// TIA Portal V16 export
// export: Created 2021-03-05T14:22:10.5832866Z, ExportSetting WithDefaults, DisplayName Totally Integrated Automation Portal, DisplayVersion V16, DisplayName TIA Portal Version Control Interface, DisplayVersion V16, DisplayName TIA Portal Openness, DisplayVersion V16, DisplayName SINAMICS Startdrive Advanced, DisplayVersion V16, DisplayName SINAMICS Startdrive G130, G150, S120, S150, SINAMICS MV, S210, DisplayVersion V16, DisplayName SINAMICS Startdrive G110M, G120, G120C, G120D, G120P, DisplayVersion V16, DisplayName STEP 7 Professional, DisplayVersion V16, DisplayName STEP 7 Safety, DisplayVersion V16, DisplayName WinCC Professional, DisplayVersion V16
FUNCTION_BLOCK "fbMain"   // FB2, LAD
{ S7_Optimized_Access := 'TRUE' }
VERSION : 0.1
// stored: AutoNumber true, IsIECCheckEnabled false, IsRetainMemResEnabled false, MemoryReserve 100, SetENOAutomatically false, UDAEnableTagReadback false
   VAR
      Room { ExternalVisible := 'False'} : Array[1.."MAX_ROOMS"] of "fbRoom";
      Config { S7_SetPoint := 'True'} : "fbConfig";
   END_VAR
   VAR_TEMP
      iRoomCount : Int;
      iRackCount : Int;
      iPos : DInt;
   END_VAR
   // Config.iNumRooms := 0;
BEGIN

REGION Network 1 (SCL)
   // bInSimulation := TRUE skips IO device configuration steps
   #Config(bInSimulation := #Config.bInSimulation);
END_REGION

REGION Network 2 (SCL)
   #Room[1].Rack[1].Fertigation.ShelvesFertigation[1].DI_Level_Switch.bStatus := "DI_Level_SW_R1S1";
   #Room[1].Rack[1].Fertigation.ShelvesFertigation[2].DI_Level_Switch.bStatus := "DI_Level_SW_R1S2";
   #Room[1].Rack[1].Fertigation.ShelvesFertigation[3].DI_Level_Switch.bStatus := "DI_Level_SW_R1S3";
   #Room[1].Rack[1].Fertigation.ShelvesFertigation[4].DI_Level_Switch.bStatus := "DI_Level_SW_R1S4";
   #Room[1].Rack[1].Fertigation.ShelvesFertigation[5].DI_Level_Switch.bStatus := "DI_Level_SW_R1S5";
   #Room[1].Rack[1].Fertigation.ShelvesFertigation[6].DI_Level_Switch.bStatus := "DI_Level_SW_R1S6";

   #Room[1].Rack[2].Fertigation.ShelvesFertigation[1].DI_Level_Switch.bStatus := "DI_Level_SW_R2S1";
   #Room[1].Rack[2].Fertigation.ShelvesFertigation[2].DI_Level_Switch.bStatus := "DI_Level_SW_R2S2";
   #Room[1].Rack[2].Fertigation.ShelvesFertigation[3].DI_Level_Switch.bStatus := "DI_Level_SW_R2S3";
   #Room[1].Rack[2].Fertigation.ShelvesFertigation[4].DI_Level_Switch.bStatus := "DI_Level_SW_R2S4";
   #Room[1].Rack[2].Fertigation.ShelvesFertigation[5].DI_Level_Switch.bStatus := "DI_Level_SW_R2S5";
   #Room[1].Rack[2].Fertigation.ShelvesFertigation[6].DI_Level_Switch.bStatus := "DI_Level_SW_R2S6";

   #Room[1].Rack[3].Fertigation.ShelvesFertigation[1].DI_Level_Switch.bStatus := "DI_Level_SW_R3S1";
   #Room[1].Rack[3].Fertigation.ShelvesFertigation[2].DI_Level_Switch.bStatus := "DI_Level_SW_R3S2";
   #Room[1].Rack[3].Fertigation.ShelvesFertigation[3].DI_Level_Switch.bStatus := "DI_Level_SW_R3S3";
   #Room[1].Rack[3].Fertigation.ShelvesFertigation[4].DI_Level_Switch.bStatus := "DI_Level_SW_R3S4";
   #Room[1].Rack[3].Fertigation.ShelvesFertigation[5].DI_Level_Switch.bStatus := "DI_Level_SW_R3S5";
   #Room[1].Rack[3].Fertigation.ShelvesFertigation[6].DI_Level_Switch.bStatus := "DI_Level_SW_R3S6";

   #Room[1].Rack[4].Fertigation.ShelvesFertigation[1].DI_Level_Switch.bStatus := "DI_Level_SW_R4S1";
   #Room[1].Rack[4].Fertigation.ShelvesFertigation[2].DI_Level_Switch.bStatus := "DI_Level_SW_R4S2";
   #Room[1].Rack[4].Fertigation.ShelvesFertigation[3].DI_Level_Switch.bStatus := "DI_Level_SW_R4S3";
   #Room[1].Rack[4].Fertigation.ShelvesFertigation[4].DI_Level_Switch.bStatus := "DI_Level_SW_R4S4";
   #Room[1].Rack[4].Fertigation.ShelvesFertigation[5].DI_Level_Switch.bStatus := "DI_Level_SW_R4S5";
   #Room[1].Rack[4].Fertigation.ShelvesFertigation[6].DI_Level_Switch.bStatus := "DI_Level_SW_R4S6";
END_REGION

REGION Network 3 (SCL)
   #Room[1].Rack[1].Fertigation.arrAI[1] := "Rack_1_Reservoir_Level";
   #Room[1].Rack[2].Fertigation.arrAI[1] := "Rack_2_Reservoir_Level";
   #Room[1].Rack[3].Fertigation.arrAI[1] := "Rack_3_Reservoir_Level";
   #Room[1].Rack[4].Fertigation.arrAI[1] := "Rack_4_Reservoir_Level";
END_REGION

REGION Network 4 (SCL): Map AI input array to all room and rack inputs
   (*
   IF #Config.Status.bDone THEN

       FOR #iRoomCount := 1 TO UINT_TO_INT("MAX_ROOMS") DO

           #iPos := 1; // input array is 1 indexed

           MOVE_BLK(IN := "GlobalAI".Room[#iRoomCount].AI[#iPos],
                    COUNT := "NUM_AI_ROOM",
                    OUT => #Room[#iRoomCount].arrAI[1]);

           #iPos += "NUM_AI_ROOM";


           FOR #iRackCount := 1 TO UINT_TO_INT("MAX_RACKS_PER_ROOM") DO

               MOVE_BLK(IN := "GlobalAI".Room[#iRoomCount].AI[#iPos],
                        COUNT := "NUM_AI_RACK",
                        OUT => #Room[#iRoomCount].Rack[#iRackCount].arrAI[1]);

               #iPos += "NUM_AI_RACK";

           END_FOR;

           #iPos += "EXTRA_AI_PER_ROOM"; // skip over unused points

       END_FOR;

   END_IF;
   *)
END_REGION

REGION Network 5 (SCL): Map DI input array to all room and rack inputs
   (*
   IF #Config.Status.bDone THEN

       FOR #iRoomCount := 1 TO UINT_TO_INT("MAX_ROOMS") DO

           #iPos := 1; // input array is 1 indexed

           (*
           MOVE_BLK(IN := "GlobalDI".Room[#iRoomCount].DI[#iPos],
                    COUNT := "MAX_DI_ROOM",
                    OUT => #Room[#iRoomCount].DI_Level_Switch.bStatus);
           *) 

           #iPos += "NUM_AI_ROOM";

           (*
           FOR #iRackCount := 1 TO UINT_TO_INT("MAX_RACKS_PER_ROOM") DO

               MOVE_BLK(IN := "GlobalDI".Room[#iRoomCount].DI[#iPos],
                        COUNT := "NUM_DI_RACK",
                        OUT => #Room[#iRoomCount].Rack[#iRackCount].arrDI[1]);

               #iPos += "NUM_AI_RACK";

           END_FOR;
           *)

           #iPos += "EXTRA_AI_PER_ROOM"; // skip over unused points

       END_FOR;

   END_IF;*)
END_REGION

REGION Network 6 (SCL): Call FBs for all configured rooms
   IF #Config.Status.bDone THEN

       FOR #iRoomCount := 1 TO #Config.iNumRooms DO

           #Room[#iRoomCount](arrAI := #Room[#iRoomCount].arrAI);

       END_FOR;

   END_IF;
END_REGION

REGION Network 7 (SCL): Combine all room and rack outputs into a single output array
   (*
   IF #Config.Status.bDone THEN

       FOR #iRoomCount := 1 TO UINT_TO_INT("MAX_ROOMS") DO

           #iPos := 1; // output array is 1 indexed

           MOVE_BLK(IN := #Room[#iRoomCount].arrDQ[1],
                    COUNT := "NUM_DQ_ROOM",
                    OUT => "GlobalDQ".Room[#iRoomCount].DQ[#iPos]);

           #iPos += "NUM_DQ_ROOM";


           FOR #iRackCount := 1 TO UINT_TO_INT("MAX_RACKS_PER_ROOM") DO

               MOVE_BLK(IN := #Room[#iRoomCount].Rack[#iRackCount].arrDQ[1],
                        COUNT := "NUM_DQ_RACK",
                        OUT => "GlobalDQ".Room[#iRoomCount].DQ[#iPos]);

               #iPos += "NUM_DQ_RACK";

           END_FOR;

           #iPos += "EXTRA_DQ_PER_ROOM"; // skip over unused points

       END_FOR;

   END_IF;
   *)
END_REGION

REGION Network 8 (SCL)
   "Rack_1_RO" := #Room[1].Rack[1].Fertigation.arrDQ[1];
   "Rack_1_Discharge" := #Room[1].Rack[1].Fertigation.arrDQ[2];

   "Rack_1_Shelf_1_Fill" := #Room[1].Rack[1].Fertigation.ShelvesFertigation[1].arrDQ[1];
   "Rack_1_Shelf_1_Drain" := #Room[1].Rack[1].Fertigation.ShelvesFertigation[1].arrDQ[2];
   "Rack_1_Shelf_2_Fill" := #Room[1].Rack[1].Fertigation.ShelvesFertigation[2].arrDQ[1];
   "Rack_1_Shelf_2_Drain" := #Room[1].Rack[1].Fertigation.ShelvesFertigation[2].arrDQ[2];
   "Rack_1_Shelf_3_Fill" := #Room[1].Rack[1].Fertigation.ShelvesFertigation[3].arrDQ[1];
   "Rack_1_Shelf_3_Drain" := #Room[1].Rack[1].Fertigation.ShelvesFertigation[3].arrDQ[2];
   "Rack_1_Shelf_4_Fill" := #Room[1].Rack[1].Fertigation.ShelvesFertigation[4].arrDQ[1];
   "Rack_1_Shelf_4_Drain" := #Room[1].Rack[1].Fertigation.ShelvesFertigation[4].arrDQ[2];
   "Rack_1_Shelf_5_Fill" := #Room[1].Rack[1].Fertigation.ShelvesFertigation[5].arrDQ[1];
   "Rack_1_Shelf_5_Drain" := #Room[1].Rack[1].Fertigation.ShelvesFertigation[5].arrDQ[2];
   "Rack_1_Shelf_6_Fill" := #Room[1].Rack[1].Fertigation.ShelvesFertigation[6].arrDQ[1];
   "Rack_1_Shelf_6_Drain" := #Room[1].Rack[1].Fertigation.ShelvesFertigation[6].arrDQ[2];

   "Rack_2_RO" := #Room[1].Rack[2].Fertigation.arrDQ[1];
   "Rack_2_Discharge" := #Room[1].Rack[2].Fertigation.arrDQ[2];

   "Rack_2_Shelf_1_Fill" := #Room[1].Rack[2].Fertigation.ShelvesFertigation[1].arrDQ[1];
   "Rack_2_Shelf_1_Drain" := #Room[1].Rack[2].Fertigation.ShelvesFertigation[1].arrDQ[2];
   "Rack_2_Shelf_2_Fill" := #Room[1].Rack[2].Fertigation.ShelvesFertigation[2].arrDQ[1];
   "Rack_2_Shelf_2_Drain" := #Room[1].Rack[2].Fertigation.ShelvesFertigation[2].arrDQ[2];
   "Rack_2_Shelf_3_Fill" := #Room[1].Rack[2].Fertigation.ShelvesFertigation[3].arrDQ[1];
   "Rack_2_Shelf_3_Drain" := #Room[1].Rack[2].Fertigation.ShelvesFertigation[3].arrDQ[2];
   "Rack_2_Shelf_4_Fill" := #Room[1].Rack[2].Fertigation.ShelvesFertigation[4].arrDQ[1];
   "Rack_2_Shelf_4_Drain" := #Room[1].Rack[2].Fertigation.ShelvesFertigation[4].arrDQ[2];
   "Rack_2_Shelf_5_Fill" := #Room[1].Rack[2].Fertigation.ShelvesFertigation[5].arrDQ[1];
   "Rack_2_Shelf_5_Drain" := #Room[1].Rack[2].Fertigation.ShelvesFertigation[5].arrDQ[2];
   "Rack_2_Shelf_6_Fill" := #Room[1].Rack[2].Fertigation.ShelvesFertigation[6].arrDQ[1];
   "Rack_2_Shelf_6_Drain" := #Room[1].Rack[2].Fertigation.ShelvesFertigation[6].arrDQ[2];


   "Rack_3_RO" := #Room[1].Rack[3].Fertigation.arrDQ[1];
   "Rack_3_Discharge" := #Room[1].Rack[3].Fertigation.arrDQ[2];

   "Rack_3_Shelf_1_Fill" := #Room[1].Rack[3].Fertigation.ShelvesFertigation[1].arrDQ[1];
   "Rack_3_Shelf_1_Drain" := #Room[1].Rack[3].Fertigation.ShelvesFertigation[1].arrDQ[2];
   "Rack_3_Shelf_2_Fill" := #Room[1].Rack[3].Fertigation.ShelvesFertigation[2].arrDQ[1];
   "Rack_3_Shelf_2_Drain" := #Room[1].Rack[3].Fertigation.ShelvesFertigation[2].arrDQ[2];
   "Rack_3_Shelf_3_Fill" := #Room[1].Rack[3].Fertigation.ShelvesFertigation[3].arrDQ[1];
   "Rack_3_Shelf_3_Drain" := #Room[1].Rack[3].Fertigation.ShelvesFertigation[3].arrDQ[2];
   "Rack_3_Shelf_4_Fill" := #Room[1].Rack[3].Fertigation.ShelvesFertigation[4].arrDQ[1];
   "Rack_3_Shelf_4_Drain" := #Room[1].Rack[3].Fertigation.ShelvesFertigation[4].arrDQ[2];
   "Rack_3_Shelf_5_Fill" := #Room[1].Rack[3].Fertigation.ShelvesFertigation[5].arrDQ[1];
   "Rack_3_Shelf_5_Drain" := #Room[1].Rack[3].Fertigation.ShelvesFertigation[5].arrDQ[2];
   "Rack_3_Shelf_6_Fill" := #Room[1].Rack[3].Fertigation.ShelvesFertigation[6].arrDQ[1];
   "Rack_3_Shelf_6_Drain" := #Room[1].Rack[3].Fertigation.ShelvesFertigation[6].arrDQ[2];

   "Rack_4_RO" := #Room[1].Rack[4].Fertigation.arrDQ[1];
   "Rack_4_Discharge" := #Room[1].Rack[4].Fertigation.arrDQ[2];

   "Rack_4_Shelf_1_Fill" := #Room[1].Rack[4].Fertigation.ShelvesFertigation[1].arrDQ[1];
   "Rack_4_Shelf_1_Drain" := #Room[1].Rack[4].Fertigation.ShelvesFertigation[1].arrDQ[2];
   "Rack_4_Shelf_2_Fill" := #Room[1].Rack[4].Fertigation.ShelvesFertigation[2].arrDQ[1];
   "Rack_4_Shelf_2_Drain" := #Room[1].Rack[4].Fertigation.ShelvesFertigation[2].arrDQ[2];
   "Rack_4_Shelf_3_Fill" := #Room[1].Rack[4].Fertigation.ShelvesFertigation[3].arrDQ[1];
   "Rack_4_Shelf_3_Drain" := #Room[1].Rack[4].Fertigation.ShelvesFertigation[3].arrDQ[2];
   "Rack_4_Shelf_4_Fill" := #Room[1].Rack[4].Fertigation.ShelvesFertigation[4].arrDQ[1];
   "Rack_4_Shelf_4_Drain" := #Room[1].Rack[4].Fertigation.ShelvesFertigation[4].arrDQ[2];
   "Rack_4_Shelf_5_Fill" := #Room[1].Rack[4].Fertigation.ShelvesFertigation[5].arrDQ[1];
   "Rack_4_Shelf_5_Drain" := #Room[1].Rack[4].Fertigation.ShelvesFertigation[5].arrDQ[2];
   "Rack_4_Shelf_6_Fill" := #Room[1].Rack[4].Fertigation.ShelvesFertigation[6].arrDQ[1];
   "Rack_4_Shelf_6_Drain" := #Room[1].Rack[4].Fertigation.ShelvesFertigation[6].arrDQ[2];
END_REGION
END_FUNCTION_BLOCK
